FUNCTION Scale : INT
VAR_INPUT
	input : INT := 0;
	in_Max : INT := 1;
	in_Min : INT := 0;
	out_Max : INT := 1;
	out_Min : INT := 0;
END_VAR
VAR
	output : INT := 0;
END_VAR


output := ((input - in_Min)/(in_Max - in_Min)*
(out_Max - out_Min)) + out_Min;

Scale := output;

END_FUNCTION

(* stored: Version 1.1.0.1, ProductVersion 3.1.4024.12
   POU Scale: Id {7feae269-51d5-4bbe-bb83-52cf51bf675f}, SpecialFunc None *)
